FUNCTION derivcvar_c: LREAL
VAR_INPUT
    state: STATE;
END_VAR

derivcvar_c := state.cvar_c;

END_FUNCTION

(* stored: ProductVersion 3.1.0.18, Version 1.1.0.1 *)
